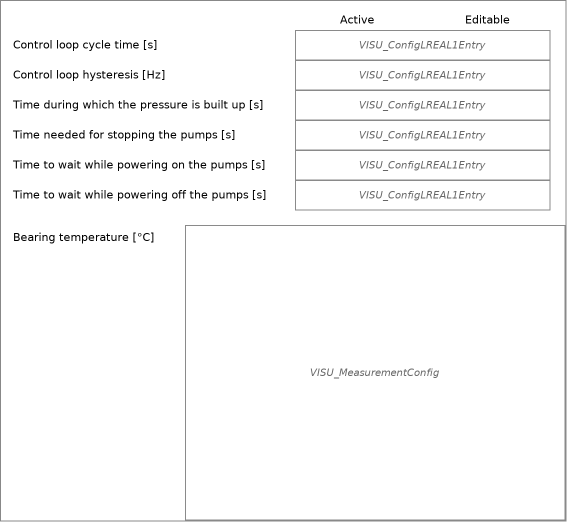
VISUALIZATION VISU_HydraulicsConfig_General  // 567x522
VAR_IN_OUT
    editable : HydraulicsConfig;
	active : HydraulicsConfig;
END_VAR
    Label (295,10 125x20), "Active"
    Label (425,10 125x20), "Editable"
    Label (10,30 250x30), "Control loop cycle time [s]"
    Label (10,60 235x30), "Control loop hysteresis [Hz]"
    Frame (295,30 255x30), tooltip "Time (in seconds) to wait after the axis has been moved"
        shows VISU_ConfigLREAL1Entry(active := active.controlCycleTime, editable := editable.controlCycleTime)
    Frame (295,60 255x30), tooltip "Time (in seconds) to wait after the axis has been moved"
        shows VISU_ConfigLREAL1Entry(active := active.controlHysteresis, editable := editable.controlHysteresis)
    Label (10,90 265x30), "Time during which the pressure is built up [s]"
    Frame (295,90 255x30), tooltip "Time (in seconds) to wait after the axis has been moved"
        shows VISU_ConfigLREAL1Entry(active := active.buildUpPressureTime, editable := editable.buildUpPressureTime)
    Label (10,120 265x30), "Time needed for stopping the pumps [s]"
    Frame (295,120 255x30), tooltip "Time (in seconds) to wait after the axis has been moved"
        shows VISU_ConfigLREAL1Entry(active := active.stoppingTime, editable := editable.stoppingTime)
    Label (10,205 170x65), "Bearing temperature [°C]"
    Frame (185,225 380x295)
        shows VISU_MeasurementConfig(active := active.bearingTemperature, editable := editable.bearingTemperature)
    Label (10,150 265x30), "Time to wait while powering on the pumps [s]"
    Frame (295,150 255x30), tooltip "Time (in seconds) to wait after the axis has been moved"
        shows VISU_ConfigLREAL1Entry(active := active.pumpsPowerOnTIme, editable := editable.pumpsPowerOnTIme)
    Label (10,180 265x30), "Time to wait while powering off the pumps [s]"
    Frame (295,180 255x30), tooltip "Time (in seconds) to wait after the axis has been moved"
        shows VISU_ConfigLREAL1Entry(active := active.pumpsPowerOffTIme, editable := editable.pumpsPowerOffTIme)
END_VISUALIZATION

(* stored: Version 1.1.0.1, ProductVersion 3.1.4019.2
   Visu VISU_HydraulicsConfig_General: Id {e8a34358-f8bd-4a20-9df8-d10ee5691768} *)
